Yaskawa INFORM job: TEST_COMARC.JBI

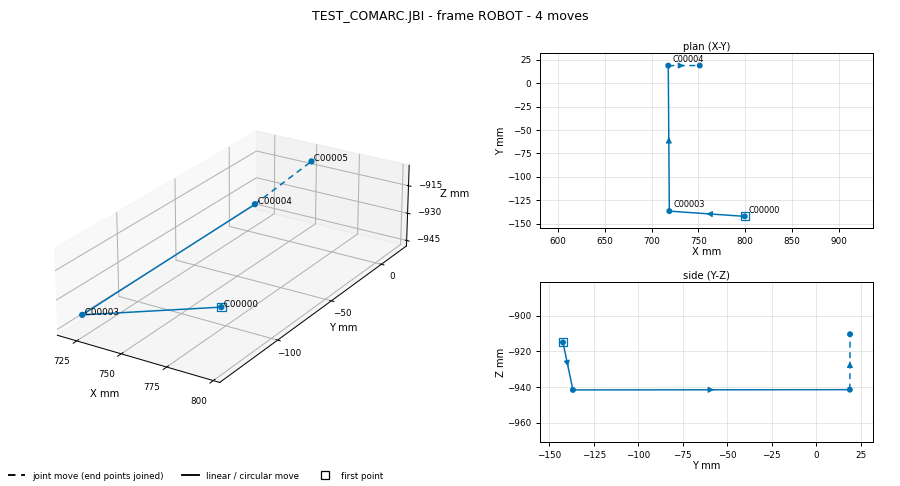
[picture p0: tool path of TEST_COMARC.JBI in frame ROBOT, 4 of 4 moves have a stored position in this frame; points joined in program order, loops and branches not executed]
/JOB
//NAME TEST_COMARC
///FOLDERNAME OTHER
//POS
///NPOS 6,6,0,0,0,0
///TOOL 0
///POSTYPE ROBOT
///RECTAN
///RCONF 1,0,0,0,0,0,0,0,0,0,0,0,0,0,0,0,0,0,0,0,0,0,0,0
C00000=799.542,-142.350,-914.891,0.4111,55.1463,-5.0636
C00001=715.811,-144.489,-922.771,-21.8407,55.3484,-23.7845
C00002=743.522,-144.489,-946.717,-21.8433,55.3458,-23.7882
C00003=718.867,-136.755,-941.610,-17.2729,48.3382,-20.1862
C00004=717.748,18.906,-941.468,-17.2684,48.3393,-20.1737
C00005=751.428,19.008,-910.305,-17.2646,48.3423,-20.1650
///RCONF 0,0,0,0,0,0,0,0,0,0,0,0,0,0,0,0,0,0,0,0,0,0,0,0
BC00000=4859.859
BC00001=4859.859
BC00002=4859.859
BC00003=4859.859
BC00004=4859.859
BC00005=4859.859
//INST
///DATE 2024/02/28 12:57
///ATTR SC,RW,RJ
////FRAME ROBOT
///GROUP1 RB1,BS1
NOP
MOVJ C00000 BC00000 VJ=0.78 PL=0
REFP 1 C00001 BC00001
REFP 2 C00002 BC00002
MOVL C00003 BC00003 V=6.7 PL=0
MACRO1 MJ#(0) ARGF1
COMM ARCON
COMARCON WEV#(1) U/D=200 L/R=10.0
MOVL C00004 BC00004 V=5.8 PL=0
COMARCOF
COMM ARCOF
MOVJ C00005 BC00005 VJ=0.78 PL=0
END
